FUNCTION_BLOCK SPLIT_AD_INTO_AQ (* this Function splits the 16 AQ (QUARTER) adapters from a AD (DWORD) *)
  (* Standard: 61499-2; Description: Copyright (c) 2026 Meisterschulen am Ostbahnhof SPDX-License-Identifier: EPL-2.0 *)
  (* Version 1.0, 2026-05-16, Franz Höpfinger, Meisterschulen am Ostbahnhof, initial API and implementation and/or initial documentation *)
  PACKAGE adapter::splitting;
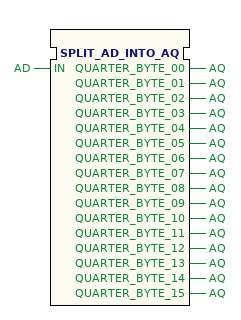
  SOCKETS
    IN : adapter::types::unidirectional::AD; (* DWORD Input *)
  END_SOCKETS
  PLUGS
    QUARTER_BYTE_00 : adapter::types::unidirectional::AQ; (* Quarter 0 *)
    QUARTER_BYTE_01 : adapter::types::unidirectional::AQ; (* Quarter 1 *)
    QUARTER_BYTE_02 : adapter::types::unidirectional::AQ; (* Quarter 2 *)
    QUARTER_BYTE_03 : adapter::types::unidirectional::AQ; (* Quarter 3 *)
    QUARTER_BYTE_04 : adapter::types::unidirectional::AQ; (* Quarter 4 *)
    QUARTER_BYTE_05 : adapter::types::unidirectional::AQ; (* Quarter 5 *)
    QUARTER_BYTE_06 : adapter::types::unidirectional::AQ; (* Quarter 6 *)
    QUARTER_BYTE_07 : adapter::types::unidirectional::AQ; (* Quarter 7 *)
    QUARTER_BYTE_08 : adapter::types::unidirectional::AQ; (* Quarter 8 *)
    QUARTER_BYTE_09 : adapter::types::unidirectional::AQ; (* Quarter 9 *)
    QUARTER_BYTE_10 : adapter::types::unidirectional::AQ; (* Quarter 10 *)
    QUARTER_BYTE_11 : adapter::types::unidirectional::AQ; (* Quarter 11 *)
    QUARTER_BYTE_12 : adapter::types::unidirectional::AQ; (* Quarter 12 *)
    QUARTER_BYTE_13 : adapter::types::unidirectional::AQ; (* Quarter 13 *)
    QUARTER_BYTE_14 : adapter::types::unidirectional::AQ; (* Quarter 14 *)
    QUARTER_BYTE_15 : adapter::types::unidirectional::AQ; (* Quarter 15 *)
  END_PLUGS
END_FUNCTION_BLOCK
